PROGRAM Ax34
VAR
	iAxisNumber : INT := E_AxisNames.Slit_3_East;
	iGroupNumber : INT := 3;
	
	stoRTrig : R_Trig;
	
	//Automatic reset on permit
	startReset : BOOL;
	resetDelay : TON;
	startDisable : BOOL;
	disableDelay : TON;
END_VAR

//Initial parameters of an Axis
IF _TaskInfo[fbGetCurTaskIndex.index].FirstCycle THEN
    //Initial default values:
    GVL.astAxes[iAxisNumber].stHomingConfig.eHomeSeq :=E_HomingRoutines.eHomeToEncPulse_BWD_FAST;
	GVL.astAxes[iAxisNumber].stHomingConfig.bGoToFwdFirst := TRUE;
	GVL.astAxes[iAxisNumber].stHomingConfig.fHomeAbsPosition:= 50;
	GVL.astAxes[iAxisNumber].stHomingConfig.fHomeMidRelativeMove:=1;
    GVL.astAxes[iAxisNumber].stHomingConfig.fHomePosition := 56.657;
    GVL.astAxes[iAxisNumber].stHomingConfig.fHomeFinishDistance := 0.0;
	GVL.astAxes[iAxisNumber].stHomingConfig.bGoToBwdFirst := TRUE;
    GVL.astAxes[iAxisNumber].stConfig.eRestorePosition := E_RestorePosition.eRestoreWithoutHome;
	GVL.astAxes[iAxisNumber].stControl.bAutoEnableDisable := TRUE;
	GVL.astAxes[iAxisNumber].stControl.tMoveFinishedDelay := T#0.1S;
	//Set which group this axis belongs to
	GVL.astAxes[iAxisNumber].stDescription.iGroupNumber := iGroupNumber;
	GVL.astAxes[iAxisNumber].Commissioning := FALSE;
	GVL.astAxes[iAxisNumber].stDescription.sUnits:= 'mm';
END_IF

GVL.astAxes[iAxisNumber].stInputs.bAllowRemoteControl:= TRUE;

//Permit
GVL.astAxes[iAxisNumber].stInputs.bPermit := SAFETY.NON_SAMPLE_PERMIT;

//Do an automatic reset on regaining permit;
IF SAFETY.NON_SAMPLE_PERMIT_R_EDGE THEN
	startReset:= TRUE;
END_IF
resetDelay(IN:= startReset, PT:= T#0.5S);
IF resetDelay.Q THEN
	startReset := FALSE;
	GVL.astAxes[iAxisNumber].stControl.bReset:= TRUE;
END_IF

//Disable axis if no permit
IF SAFETY.STOP_NON_SAMPLE_MOTION THEN
	startDisable := TRUE;
END_IF
disableDelay(IN:= startDisable, PT:= T#1S);
IF disableDelay.Q THEN
	startDisable:= FALSE;
	GVL.astAxes[iAxisNumber].stControl.bEnable:= FALSE;
END_IF

//Safety stop motion
IF SAFETY.STOP_NON_SAMPLE_MOTION THEN
	GVL.astAxes[iAxisNumber].stControl.bHalt:= TRUE;
END_IF

stoRTrig(CLK:=GVL.astAxes[iAxisNumber].stStatus.bSTOActive);
IF stoRTrig.Q THEN
	GVL.astAxes[iAxisNumber].stControl.bReset:= TRUE;
END_IF




//Define ACTIONS() or write exclusive code for an specific axis.
(*Eg. Stop when temperature reaches certain values, reduce speed if  a signal is activated, etc.
Eg. GVL.astAxes[x].stControl.bInterlockFwd := NOT bInterlockFwdOK;*)

END_PROGRAM

(* stored: Version 1.1.0.1, ProductVersion 3.1.4026.18
   POU Ax34: Id {95a34dbb-cff1-401f-bf17-ef76c3c117e5}, SpecialFunc None *)
